FUNCTION_BLOCK FB_Cylinder
VAR
	_bExtended, _bRetracted	: BOOL;
	refExtendOut			: REFERENCE TO BOOL;
	refRetractOut			: REFERENCE TO BOOL;
END_VAR

// The cylinder is edge-free: the sensor image is refreshed every cycle and the outputs
// are held by whichever of Extend()/Retract() was called last.
Cyclic();

METHOD FB_init : BOOL
VAR_INPUT
	bInitRetains	: BOOL;
	bInCopyCode		: BOOL;
	refExtendOut	: REFERENCE TO BOOL;
	refRetractOut	: REFERENCE TO BOOL;
END_VAR
THIS^.refExtendOut REF= refExtendOut;
THIS^.refRetractOut REF= refRetractOut;
FB_init := TRUE;
END_METHOD

METHOD Extend : BOOL
VAR
END_VAR
refExtendOut := TRUE;
refRetractOut := FALSE;
Extend := TRUE;
END_METHOD

METHOD Retract : BOOL
VAR
END_VAR
refExtendOut := FALSE;
refRetractOut := TRUE;
Retract := TRUE;
END_METHOD

METHOD Cyclic
VAR
END_VAR
_bExtended := GVL_Io.bSensorExtended;
_bRetracted := GVL_Io.bSensorRetracted;
END_METHOD

PROPERTY bIsExtended : BOOL
GET
bIsExtended := _bExtended;
END_GET
END_PROPERTY

PROPERTY bIsRetracted : BOOL
GET
bIsRetracted := _bRetracted;
END_GET
END_PROPERTY

END_FUNCTION_BLOCK

(* stored: Version 1.1.0.1, ProductVersion 3.1.4024.12
   POU FB_Cylinder: Id {41f79a40-cd4e-4358-970b-e801671e1e8d}, SpecialFunc None
   Method FB_init: Id {6097e33e-405f-41ad-9501-d14f45c207c2}
   Method Extend: Id {12cc0988-1857-48cf-a28a-4fddaf18dda0}
   Method Retract: Id {82ae731f-7528-49aa-bdc1-4bc5ade12f80}
   Method Cyclic: Id {452233ea-0599-45d3-9a25-18bcf402609e}
   Property bIsExtended: Id {a74466b3-f26f-450e-846b-2e80bc9d329a}
   Get Get: Id {51917955-a8bd-429d-811b-67d394dbb16b}
   Property bIsRetracted: Id {1b734660-6b74-4853-a2cb-d0deb6e7a890}
   Get Get: Id {6bf331d1-d8f9-4d84-86a9-5cb027044fe0} *)
